// TIA Portal V19 export
VAR_GLOBAL   // PLC tag table "MTR"
END_VAR
